PROGRAM P_Station
VAR
	_stParameter:				ST_StationParameter;
	_stHandshake:				ST_StationHandshake;
	
	_fbTakeLoad:				FB_StationTakeLoad;// 取料站
	_fbDismantling_L2:			FB_StationDismantling;// 线体2 拆解站 
	_fbDismantling_L3:			FB_StationDismantling;// 线体3 拆解站 
	_fbLine0Load:				FB_StationLine0Load;// 线体0 上料站
	_fbLine0Buffer:				FB_StationLine0Buffer;// 线体0 缓存站
	_fbLineLoad_L1:				FB_StationLineLoad;// 线体1 上料站
	_fbLineLoad_L3:				FB_StationLineLoad;// 线体3 上料站
	_fbUnloadUc_L2:				FB_StationUnloadUc;// 线体2 下UC
	_fbUnloadUc_L3:				FB_StationUnloadUc;// 线体3 下UC
	_fbUnloadElevator_L2:		FB_StationUnloadElevator;// 线体2 下工装
	_fbUnloadElevator_L3:		FB_StationUnloadElevator;// 线体3 下工装
	_fbUnloadLineUc:			FB_StationUnloadLine;//下UC 线体
	_fbUnloadLineElevator:		FB_StationUnloadLine;// 下工装线体
	_fbStationUnLoadUc_311:		FB_StationUnLoadUc_311;// 下UC 模组
		
	_vArrFbCylinder:			ARRAY[0..10] OF FB_Cylinder;// 虚拟气缸
	_vArrCylinder:				ARRAY[0..10] OF ST_Cylinder;// 虚拟气缸
	_vArrCylinderData:			ARRAY[0..10] OF ST_CylinderData;// 虚拟气缸
	_i:							INT;
	_bFistRun:					BOOL:=true;
END_VAR

GVL.stSetting.eTakeMode:=M_LoadPriority(_stParameter,GVL_Data.stRecipe);
IF _bFistRun THEN
	A_Info();
	_bFistRun:=FALSE;
END_IF


A_Handshake();// 交握

A_Virtual();// 虚拟硬件



A_TakeLoad();// 取料站

A_Dismantling_L2();// 拆解站

A_Dismantling_L3();// 拆解站

A_Line0Buffer();// 线体0 上料缓存

A_Line0Load();// 线体0 上料站

A_LineLoad_L1();// 线体1 上料

A_LineLoad_L3();// 线体3 上料

A_UnloadElevator_L2();// 线体2 下工装

A_UnloadElevator_L3();// 线体3 下工装

A_UnloadLineElevator();// 下工装 流线

A_UnLoadUc_311();// 下UC模组  紧311使用

A_UnloadLineUc();// 下UC 流线 311以为下料程序

A_UnloadUc_L2();// 线体2下UC 311以外下料程序

A_UnloadUc_L3();// 线体3 下UC 311以为下料程序

ACTION A_Dismantling_L2:
_stParameter.stLine2Dismantling.bPalletCheck1:=GVL.I.bLine2PalletCheck1;
_stParameter.stLine2Dismantling.bPalletCheck2:=GVL.I.bLine2PalletCheck2;
_stParameter.stLine2Dismantling.bPalletCheck3:=GVL.I.bLine2PalletCheck3;
_stParameter.stLine2Dismantling.fbLateral1 REF=G_arrFbCylinder[E_Cylinder.Line2OpenLateral1];
_stParameter.stLine2Dismantling.fbLateral2 REF=G_arrFbCylinder[E_Cylinder.Line2OpenLateral2];
_stParameter.stLine2Dismantling.fbLift REF= G_arrFbCylinder[E_Cylinder.Line2Lift];
_stParameter.stLine2Dismantling.fbPrevent REF= G_arrFbCylinder[E_Cylinder.Line2Prevent];
_stParameter.stLine2Dismantling.fbRotate REF= G_arrFbCylinder[E_Cylinder.Line2OpenRotate];
_stParameter.stLine2Dismantling.fbStandard1 REF= G_arrFbCylinder[E_Cylinder.Line2Standard1];
_stParameter.stLine2Dismantling.fbStandard2 REF= G_arrFbCylinder[E_Cylinder.Line2Standard2];
_stParameter.stLine2Dismantling.bClose:=GVL_Data.stRecipe.eLineClose=E_LineClose.Line2;
_stParameter.stLine2Dismantling.bCloseUnloadElevator:=FALSE;

_fbDismantling_L2(
	Enable:=TRUE,
	System:=G_stSystem , 
	Station:=G_arrStation[E_Station.Line2Dismantling] , 
	Error:=G_stError , 
	Setting:=GVL.stSetting , 
	Recipe:=GVL_Data.stRecipe , 
	Parameter:=_stParameter.stLine2Dismantling);
END_ACTION

ACTION A_Dismantling_L3:
_stParameter.stLine3Dismantling.bPalletCheck1:=GVL.I.bLine3OpenCheck1;
_stParameter.stLine3Dismantling.bPalletCheck2:=GVL.I.bLine3OpenCheck2;
_stParameter.stLine3Dismantling.bPalletCheck3:=GVL.I.bLine3OpenCheck3;
_stParameter.stLine3Dismantling.fbLateral1 REF=G_arrFbCylinder[E_Cylinder.Line3OpenLateral1];
_stParameter.stLine3Dismantling.fbLateral2 REF=G_arrFbCylinder[E_Cylinder.Line3OpenLateral2];
_stParameter.stLine3Dismantling.fbLift REF= G_arrFbCylinder[E_Cylinder.Line3OpenLift];
_stParameter.stLine3Dismantling.fbPrevent REF= G_arrFbCylinder[E_Cylinder.Line3OpenPrevent];
_stParameter.stLine3Dismantling.fbRotate REF= G_arrFbCylinder[E_Cylinder.Line3OpenRotate];
_stParameter.stLine3Dismantling.fbStandard1 REF= G_arrFbCylinder[E_Cylinder.Line3Standard1];
_stParameter.stLine3Dismantling.fbStandard2 REF= G_arrFbCylinder[E_Cylinder.Line3Standard2];
_stParameter.stLine3Dismantling.bClose:=GVL_Data.stRecipe.eLineClose=E_LineClose.Line3;
_stParameter.stLine3Dismantling.bCloseUnloadElevator:=FALSE;

_fbDismantling_L3(
	Enable:=TRUE,
	System:=G_stSystem , 
	Station:=G_arrStation[E_Station.Line3Dismantling] , 
	Error:=G_stError , 
	Setting:=GVL.stSetting , 
	Recipe:=GVL_Data.stRecipe , 
	Parameter:=_stParameter.stLine3Dismantling);
END_ACTION

ACTION A_Handshake:
_stParameter.stLine0Load.stHandshake.bRequestLine0Load:=_stParameter.stLine0Buffer.stHandshake.bRequestLine0Load;

_stParameter.stLine0Buffer.stHandshake.bRequestLine0Buffer_T:=_stParameter.stTakeLoad.stHandshake.bRequestLine0Buffer_T0;
_stParameter.stLine0Buffer.stHandshake.bResponseLine0Buffer:=_stParameter.stLine0Load.stHandshake.bResponseLine0Buffer;

_stParameter.stLine1Load.stHandshake.bRequestLineLoad_D:=_stParameter.stLine2Dismantling.stHandshake.bRequestLineLoad_D;
_stParameter.stLine1Load.stHandshake.bRequestLineLoad_P:=_stParameter.stTakeLoad.stHandshake.bRequestLineLoad_P1;
_stParameter.stLine1Load.stHandshake.bRequestLineLoad_T:=_stParameter.stTakeLoad.stHandshake.bRequestLineLoad_T1;
_stParameter.stLine1Load.stHandshake.bRequestTake_P_M:=FALSE;
_stParameter.stLine1Load.stHandshake.bResponseMachine_P:=FALSE;

_stParameter.stLine2UnloadElevator.stHandshake.bRequestElevator:=_stParameter.stLine2Dismantling.stHandshake.bRequestElevator;
_stParameter.stLine2UnloadElevator.stHandshake.bResponseElevator:=_stParameter.stUnloadLineElevator.stHandshake.bResponseUnladLine2;

_stParameter.stLine2UnloadUc.stHandshake.bResponseUnladLine:=_stParameter.stUnloadLineUc.stHandshake.bResponseUnladLine2;

_stParameter.stLine3Load.stHandshake.bRequestLineLoad_D:=_stParameter.stLine3Dismantling.stHandshake.bRequestLineLoad_D;
_stParameter.stLine3Load.stHandshake.bRequestLineLoad_P:=_stParameter.stTakeLoad.stHandshake.bRequestLineLoad_P3;
_stParameter.stLine3Load.stHandshake.bRequestLineLoad_T:=_stParameter.stTakeLoad.stHandshake.bRequestLineLoad_T3;
_stParameter.stLine3Load.stHandshake.bRequestTake_P_M:=FALSE;
_stParameter.stLine3Load.stHandshake.bResponseMachine_P:=FALSE;

_stParameter.stLine3UnloadElevator.stHandshake.bRequestElevator:=_stParameter.stLine3Dismantling.stHandshake.bRequestElevator;
_stParameter.stLine3UnloadElevator.stHandshake.bResponseElevator:=_stParameter.stUnloadLineElevator.stHandshake.bResponseUnladLine3;

_stParameter.stLine3UnloadUc.stHandshake.bResponseUnladLine:=_stParameter.stUnloadLineUc.stHandshake.bResponseUnladLine3;

_stParameter.stTakeLoad.stHandshake.bResponseTake_P1:=_stParameter.stLine1Load.stHandshake.bResponseTake_P;
_stParameter.stTakeLoad.stHandshake.bResponseTake_P3:=_stParameter.stLine3Load.stHandshake.bResponseTake_P;
_stParameter.stTakeLoad.stHandshake.bResponseTake_T0:=_stParameter.stLine0Buffer.stHandshake.bResponseTake_T;
_stParameter.stTakeLoad.stHandshake.bResponseTake_T1:=_stParameter.stLine1Load.stHandshake.bResponseTake_T;
_stParameter.stTakeLoad.stHandshake.bResponseTake_T3:=_stParameter.stLine3Load.stHandshake.bResponseTake_T;

_stParameter.stUnloadLineElevator.stHandshake.bRequestUnloadLine2:=_stParameter.stLine2UnloadElevator.stHandshake.bRequestUnline;
_stParameter.stUnloadLineElevator.stHandshake.bRequestUnloadLine3:=_stParameter.stLine3UnloadElevator.stHandshake.bRequestUnline;

_stParameter.stUnloadLineUc.stHandshake.bRequestUnloadLine2:=_stParameter.stLine2UnloadUc.stHandshake.bRequestUnloadLine;
_stParameter.stUnloadLineUc.stHandshake.bRequestUnloadLine3:=_stParameter.stLine3UnloadUc.stHandshake.bRequestUnloadLine;

_stParameter.stLine2Dismantling.stHandshake.bResponseDismantling_D:=_stParameter.stLine1Load.stHandshake.bResponseDismantling_D;
_stParameter.stLine2Dismantling.stHandshake.bResponseDismantling_E:=_stParameter.stLine2UnloadElevator.stHandshake.bResponseDismantling_E;
_stParameter.stLine3Dismantling.stHandshake.bResponseDismantling_D:=_stParameter.stLine3Load.stHandshake.bResponseDismantling_D;
_stParameter.stLine3Dismantling.stHandshake.bResponseDismantling_E:=_stParameter.stLine3UnloadElevator.stHandshake.bResponseDismantling_E;

IF GVL_Data.stRecipe.eMachineType =E_MachineType.RH311 OR GVL_Data.stRecipe.eMachineType =E_MachineType.LH311 THEN
	_stParameter.stUnloadUc_311.stHandshake.bRequestUc_L2:=_stParameter.stLine2Dismantling.stHandshake.bRequestUc;
	_stParameter.stUnloadUc_311.stHandshake.bRequestUc_L3:=_stParameter.stLine3Dismantling.stHandshake.bRequestUc;
	_stParameter.stLine2Dismantling.stHandshake.bResponseDismantling_Uc:=_stParameter.stUnloadUc_311.stHandshake.bResponseDismantling_Uc_L2;
	_stParameter.stLine3Dismantling.stHandshake.bResponseDismantling_Uc:=_stParameter.stUnloadUc_311.stHandshake.bResponseDismantling_Uc_L3;
ELSE
	_stParameter.stLine2UnloadUc.stHandshake.bRequestUc:=_stParameter.stLine2Dismantling.stHandshake.bRequestUc;
	_stParameter.stLine3UnloadUc.stHandshake.bRequestUc:=_stParameter.stLine3Dismantling.stHandshake.bRequestUc;
	_stParameter.stLine2Dismantling.stHandshake.bResponseDismantling_Uc:=_stParameter.stLine2UnloadUc.stHandshake.bResponseDismantling_Uc;
	_stParameter.stLine3Dismantling.stHandshake.bResponseDismantling_Uc:=_stParameter.stLine3UnloadUc.stHandshake.bResponseDismantling_Uc;
END_IF
END_ACTION

ACTION A_Info:
_i:=E_Station.Line0Load;
G_arrStation[_i].arrName[E_Language.Chinese]:="主流线上料工站";
G_arrStation[_i].arrName[E_Language.English]:="Line0Load";
G_arrStation[_i].arrName[E_Language.Vietnamese]:="Trạm vật liệu dòng chính";

_i:=E_Station.Line0Buffer;
G_arrStation[_i].arrName[E_Language.Chinese]:="主流线缓存工站";
G_arrStation[_i].arrName[E_Language.English]:="Line0Buffer";
G_arrStation[_i].arrName[E_Language.Vietnamese]:="Trạm bộ nhớ nhớ đường chính";

_i:=E_Station.TakeLoad;
G_arrStation[_i].arrName[E_Language.Chinese]:="上料取料工站";
G_arrStation[_i].arrName[E_Language.English]:="TakeLoad";
G_arrStation[_i].arrName[E_Language.Vietnamese]:="Nhà ga ăn uống";

_i:=E_Station.Line3Load;
G_arrStation[_i].arrName[E_Language.Chinese]:="流线3上料工站";
G_arrStation[_i].arrName[E_Language.English]:="Line3Load";
G_arrStation[_i].arrName[E_Language.Vietnamese]:="Trạm sạc 3 dòng";

_i:=E_Station.Line1Load;
G_arrStation[_i].arrName[E_Language.Chinese]:="流线2上料工站";
G_arrStation[_i].arrName[E_Language.English]:="Line1Load";
G_arrStation[_i].arrName[E_Language.Vietnamese]:="Trạm lên men dòng 2";

_i:=E_Station.Line2Dismantling;
G_arrStation[_i].arrName[E_Language.Chinese]:="流线2拆解工站";
G_arrStation[_i].arrName[E_Language.English]:="Line2Dismantling";
G_arrStation[_i].arrName[E_Language.Vietnamese]:="Trạm tháo dỡ dòng 2";

_i:=E_Station.Line3Dismantling;
G_arrStation[_i].arrName[E_Language.Chinese]:="流线3拆解工站";
G_arrStation[_i].arrName[E_Language.English]:="Line3Dismantling";
G_arrStation[_i].arrName[E_Language.Vietnamese]:="Trạm tháo dỡ dòng 3";

_i:=E_Station.Line2UnloadElevator;
G_arrStation[_i].arrName[E_Language.Chinese]:="线体2下工装";
G_arrStation[_i].arrName[E_Language.English]:="Line2UnloadElevator";
G_arrStation[_i].arrName[E_Language.Vietnamese]:="Thiết bị dây chuyền 2";

_i:=E_Station.Line3UnloadElevator;
G_arrStation[_i].arrName[E_Language.Chinese]:="线体3下工装";
G_arrStation[_i].arrName[E_Language.English]:="Line3UnloadElevator";
G_arrStation[_i].arrName[E_Language.Vietnamese]:="Dây số 3 dưới công cụ";

_i:=E_Station.Line2UnloadUc;
G_arrStation[_i].arrName[E_Language.Chinese]:="线体2 下UC";
G_arrStation[_i].arrName[E_Language.English]:="Line2UnloadUc";
G_arrStation[_i].arrName[E_Language.Vietnamese]:="Máy dò 2 ở UC";

_i:=E_Station.Line3UnloadUc;
G_arrStation[_i].arrName[E_Language.Chinese]:="线体3 下UC";
G_arrStation[_i].arrName[E_Language.English]:="Line3UnloadUc";
G_arrStation[_i].arrName[E_Language.Vietnamese]:="Máy dò 3 ở UC";

_i:=E_Station.UnloadLineUc;
G_arrStation[_i].arrName[E_Language.Chinese]:="下UC 线体";
G_arrStation[_i].arrName[E_Language.English]:="UnloadLineUc";
G_arrStation[_i].arrName[E_Language.Vietnamese]:="Ống dẫn dưới UC";

_i:=E_Station.UnloadLineElevator;
G_arrStation[_i].arrName[E_Language.Chinese]:="下工装 线体";
G_arrStation[_i].arrName[E_Language.English]:="UnloadLineElevator";
G_arrStation[_i].arrName[E_Language.Vietnamese]:="Thiết bị dây";

_i:=E_Station.UnloadUc_311;
G_arrStation[_i].arrName[E_Language.Chinese]:="下UC模组";
G_arrStation[_i].arrName[E_Language.English]:="UnloadUc_311";
G_arrStation[_i].arrName[E_Language.Vietnamese]:="Mô-đun dưới UC";
END_ACTION

ACTION A_Line0Buffer:

_stParameter.stLine0Buffer.bPlace:=GVL.I.bLine0Place;


_fbLine0Buffer(
	Enable:=TRUE,
	System:=G_stSystem , 
	Station:=G_arrStation[E_Station.Line0Buffer] , 
	Error:=G_stError , 
	Setting:=GVL.stSetting , 
	Recipe:=GVL_Data.stRecipe , 
	Parameter:=_stParameter.stLine0Buffer);
END_ACTION

ACTION A_Line0Load:
_stParameter.stLine0Load.bPartCheck:=GVL.I.bLine0Part;
_stParameter.stLine0Load.bPreventCheck:=GVL.I.bLine0Prevent;
_stParameter.stLine0Load.fbPart REF= G_arrFbCylinder[E_Cylinder.Line0Part];
_stParameter.stLine0Load.fbPrevent REF= G_arrFbCylinder[E_Cylinder.Line0Prevent];

_fbLine0Load(
	Enable:=TRUE,
	System:=G_stSystem , 
	Station:=G_arrStation[E_Station.Line0Load] , 
	Error:=G_stError , 
	Setting:=GVL.stSetting , 
	Recipe:=GVL_Data.stRecipe , 
	Parameter:=_stParameter.stLine0Load);
END_ACTION

ACTION A_LineLoad_L1:
_stParameter.stLine1Load.bIsClosed:=GVL_Data.stRecipe.eLoadClose=E_LoadClose.Line1;
_stParameter.stLine1Load.bIsPlacing:=GVL.stSetting.eTakeModeBuffer=E_TakeMode.Place1;
_stParameter.stLine1Load.bIsTaking:=GVL.stSetting.eTakeModeBuffer=E_TakeMode.Take1;
_stParameter.stLine1Load.bPalletCheck1:=GVL.I.bLine1PalletCheck1;
_stParameter.stLine1Load.bPalletCheck2:=GVL.I.bLine1PalletCheck2;
_stParameter.stLine1Load.bPalletCheck3:=GVL.I.bLine1PalletCheck3;
_stParameter.stLine1Load.fbAdjust1 REF= G_arrFbCylinder[E_Cylinder.Line1Adjust1];
_stParameter.stLine1Load.fbElevator REF= G_arrFbCylinder[E_Cylinder.Line1Elevator];
_stParameter.stLine1Load.fbLift REF= G_arrFbCylinder[E_Cylinder.Line1Lift];
_stParameter.stLine1Load.fbPrevent REF= G_arrFbCylinder[E_Cylinder.Line1Prevent];
_stParameter.stLine1Load.fbRotate REF= G_arrFbCylinder[E_Cylinder.Line1Rotate];
_stParameter.stLine1Load.bManualLoad:=FALSE;
_fbLineLoad_L1(
	Enable:=true,
	System:=G_stSystem , 
	Station:=G_arrStation[E_Station.Line1Load] , 
	Error:=G_stError , 
	Setting:=GVL.stSetting , 
	Recipe:=GVL_Data.stRecipe , 
	Parameter:=_stParameter.stLine1Load);
END_ACTION

ACTION A_LineLoad_L3:
_stParameter.stLine3Load.bIsClosed:=FALSE;
_stParameter.stLine3Load.bIsPlacing:=GVL.stSetting.eTakeModeBuffer=E_TakeMode.Place3Load;
_stParameter.stLine3Load.bIsTaking:=GVL.stSetting.eTakeModeBuffer=E_TakeMode.Take3Load;
_stParameter.stLine3Load.bPalletCheck1:=GVL.I.bLine3PalletCheck1;
_stParameter.stLine3Load.bPalletCheck2:=GVL.I.bLine3PalletCheck2;
_stParameter.stLine3Load.bPalletCheck3:=GVL.I.bLine3PalletCheck3;
_stParameter.stLine3Load.fbAdjust1 REF= _vArrFbCylinder[0];
_stParameter.stLine3Load.fbElevator REF=_vArrFbCylinder[1];
_stParameter.stLine3Load.fbLift REF= G_arrFbCylinder[E_Cylinder.Line3LoadLift];
_stParameter.stLine3Load.fbPrevent REF= G_arrFbCylinder[E_Cylinder.Line3LoadPrevent];
_stParameter.stLine3Load.fbRotate REF= G_arrFbCylinder[E_Cylinder.Line3LoadRotate];
_stParameter.stLine3Load.bManualLoad:=FALSE;

_fbLineLoad_L3(
	Enable:=TRUE,
	System:=G_stSystem , 
	Station:=G_arrStation[E_Station.Line3Load] , 
	Error:=G_stError , 
	Setting:=GVL.stSetting , 
	Recipe:=GVL_Data.stRecipe , 
	Parameter:=_stParameter.stLine3Load);
END_ACTION

ACTION A_TakeLoad:
_stParameter.stTakeLoad.fbTakeClamp REF= G_arrFbCylinder[E_Cylinder.TakeClamp];
_stParameter.stTakeLoad.fbTakeLift1 REF= G_arrFbCylinder[E_Cylinder.TakeLift1];
_stParameter.stTakeLoad.fbTakeLift2 REF= G_arrFbCylinder[E_Cylinder.TakeLift2];
_stParameter.stTakeLoad.fbTakeY REF= G_arrFbAxis[E_Axis.TakeY];
_stParameter.stTakeLoad.fbTakeZ REF= G_arrFbAxis[E_Axis.TakeZ];

_fbTakeLoad(
	Enable:=TRUE,
	System:=G_stSystem , 
	Station:=G_arrStation[E_Station.TakeLoad] , 
	Error:=G_stError , 
	Setting:=GVL.stSetting , 
	Recipe:=GVL_Data.stRecipe , 
	Parameter:=_stParameter.stTakeLoad);
END_ACTION

ACTION A_UnloadElevator_L2:
_stParameter.stLine2UnloadElevator.bFrockElevator1NoneCheck:=GVL.I.bFrockElevator1NoneCheck;
_stParameter.stLine2UnloadElevator.fbFrockElevator REF= G_arrFbCylinder[E_Cylinder.FrockElevator1];
_stParameter.stLine2UnloadElevator.fbFrockPush REF= G_arrFbCylinder[E_Cylinder.FrockPush1];
_stParameter.stLine2UnloadElevator.fbFrockRotateDown REF= G_arrFbCylinder[E_Cylinder.FrockRotateDown1];
_stParameter.stLine2UnloadElevator.bManualUnload:=FALSE;


_fbUnloadElevator_L2(
	Enable:=TRUE,
	System:=G_stSystem , 
	Station:=G_arrStation[E_Station.Line2UnloadElevator] , 
	Error:=G_stError , 
	Setting:=GVL.stSetting , 
	Recipe:=GVL_Data.stRecipe , 
	Parameter:=_stParameter.stLine2UnloadElevator);
END_ACTION

ACTION A_UnloadElevator_L3:

_stParameter.stLine3UnloadElevator.bFrockElevator1NoneCheck:=GVL.I.bFrockElevator2NoneCheck;
_stParameter.stLine3UnloadElevator.fbFrockElevator REF= G_arrFbCylinder[E_Cylinder.FrockElevator2];
_stParameter.stLine3UnloadElevator.fbFrockPush REF= G_arrFbCylinder[E_Cylinder.FrockPush2];
_stParameter.stLine3UnloadElevator.fbFrockRotateDown REF= G_arrFbCylinder[E_Cylinder.FrockRotateDown2];
_stParameter.stLine3UnloadElevator.bManualUnload:=FALSE;

_fbUnloadElevator_L3(
	Enable:=TRUE,
	System:=G_stSystem , 
	Station:=G_arrStation[E_Station.Line3UnloadElevator] , 
	Error:=G_stError , 
	Setting:=GVL.stSetting , 
	Recipe:=GVL_Data.stRecipe , 
	Parameter:=_stParameter.stLine3UnloadElevator);
END_ACTION

ACTION A_UnloadLineElevator:
_stParameter.stUnloadLineElevator.bBeltDone:=GVL.I.bFrockBeltDone;
_stParameter.stUnloadLineElevator.bBeltNoneCheck:=GVL.I.bFrockBeltNoneCheck3;
_stParameter.stUnloadLineElevator.bCheck1:=GVL.I.bFrockBeltNoneCheck1;
_stParameter.stUnloadLineElevator.bCheck2:=GVL.I.bFrockBeltNoneCheck2;
_stParameter.stUnloadLineElevator.fbDrive REF= G_arrFbCylinder[E_Cylinder.FrockBelt];
_stParameter.stUnloadLineElevator.fbLineAxis REF= GVL.arrFbLine[E_Line.UnloadElevator];
_stParameter.stUnloadLineElevator.bManualUnload:=FALSE;

_fbUnloadLineElevator(
	Enable:=TRUE,
	System:=G_stSystem , 
	Station:=G_arrStation[E_Station.UnloadLineElevator] , 
	Error:=G_stError , 
	Setting:=GVL.stSetting , 
	Recipe:=GVL_Data.stRecipe , 
	Parameter:=_stParameter.stUnloadLineElevator);
END_ACTION

ACTION A_UnloadLineUc:
_stParameter.stUnloadLineUc.bBeltDone:=GVL.I.bUcBeltDone;
_stParameter.stUnloadLineUc.bBeltNoneCheck:=GVL.I.bUcBeltNoneCheck;
_stParameter.stUnloadLineUc.bCheck1:=GVL.I.bUcCheck2;
_stParameter.stUnloadLineUc.bCheck2:=GVL.I.bUcCheck3;
_stParameter.stUnloadLineUc.fbDrive REF= G_arrFbCylinder[E_Cylinder.UcDrive];
_stParameter.stUnloadLineUc.fbLineAxis REF= GVL.arrFbLine[E_Line.UnloadUC];
_stParameter.stUnloadLineUc.bManualUnload:=FALSE;

_fbUnloadLineUc(
	Enable:=NOT(GVL_Data.stRecipe.eMachineType=E_MachineType.LH311 OR GVL_Data.stRecipe.eMachineType=E_MachineType.RH311),
	System:=G_stSystem , 
	Station:=G_arrStation[E_Station.UnloadLineUc] , 
	Error:=G_stError , 
	Setting:=GVL.stSetting , 
	Recipe:=GVL_Data.stRecipe , 
	Parameter:=_stParameter.stUnloadLineUc);
END_ACTION

ACTION A_UnLoadUc_311:
_stParameter.stUnloadUc_311.bUcCheck1:=GVL.I.bUcCheck1;
_stParameter.stUnloadUc_311.fbAxisY REF= G_arrFbAxis[E_Axis.UC_Y];
_stParameter.stUnloadUc_311.fbClamp REF= G_arrFbCylinder[E_Cylinder.UcClamp];
_stParameter.stUnloadUc_311.fbLift REF= G_arrFbCylinder[E_Cylinder.UcLift];
_stParameter.stUnloadUc_311.fbSwing REF= G_arrFbCylinder[E_Cylinder.UcSwing];

_fbStationUnLoadUc_311(
	Enable:=GVL_Data.stRecipe.eMachineType=E_MachineType.LH311 OR GVL_Data.stRecipe.eMachineType=E_MachineType.RH311,
	System:=G_stSystem , 
	Station:=G_arrStation[E_Station.UnloadUc_311] , 
	Error:=G_stError , 
	Setting:=GVL.stSetting , 
	Recipe:=GVL_Data.stRecipe , 
	Parameter:=_stParameter.stUnloadUc_311);
END_ACTION

ACTION A_UnloadUc_L2:
_stParameter.stLine2UnloadUc.fbClamp REF= G_arrFbCylinder[E_Cylinder.UcClamp1];
_stParameter.stLine2UnloadUc.fbLift REF= G_arrFbCylinder[E_Cylinder.UcLift1];
_stParameter.stLine2UnloadUc.fbRotate REF= G_arrFbCylinder[E_Cylinder.UcRotate1];

_fbUnloadUc_L2(
	Enable:=NOT(GVL_Data.stRecipe.eMachineType=E_MachineType.LH311 OR GVL_Data.stRecipe.eMachineType=E_MachineType.RH311),
	System:=G_stSystem , 
	Station:=G_arrStation[E_Station.Line2UnloadUc] , 
	Error:=G_stError , 
	Setting:=GVL.stSetting , 
	Recipe:=GVL_Data.stRecipe , 
	Parameter:=_stParameter.stLine2UnloadUc);
END_ACTION

ACTION A_UnloadUc_L3:
_stParameter.stLine3UnloadUc.fbClamp REF= G_arrFbCylinder[E_Cylinder.UcClamp2];
_stParameter.stLine3UnloadUc.fbLift REF= G_arrFbCylinder[E_Cylinder.UcLift2];
_stParameter.stLine3UnloadUc.fbRotate REF= G_arrFbCylinder[E_Cylinder.UcRotate2];

	
_fbUnloadUc_L3(
	Enable:=NOT(GVL_Data.stRecipe.eMachineType=E_MachineType.LH311 OR GVL_Data.stRecipe.eMachineType=E_MachineType.RH311),
	System:=G_stSystem , 
	Station:=G_arrStation[E_Station.Line3UnloadUc] , 
	Error:=G_stError , 
	Setting:=GVL.stSetting , 
	Recipe:=GVL_Data.stRecipe , 
	Parameter:=_stParameter.stLine3UnloadUc);
END_ACTION

ACTION A_Virtual:
FOR _i:=0 TO 10 BY 1 DO
	_vArrCylinder[_i].stInput.bHome:=_vArrCylinder[_i].stOutput.bHome;
	_vArrCylinder[_i].stInput.bWork:=_vArrCylinder[_i].stOutput.bWork;
	_vArrFbCylinder[_i](System:=G_stSystem , Cylinder:=_vArrCylinder[_i] , Data:=_vArrCylinderData[_i] , Error:=G_stError );
END_FOR
END_ACTION

METHOD M_LoadPriority : E_TakeMode
VAR_INPUT
	Parameter:		 REFERENCE TO ST_StationParameter;
	Recipe:			 REFERENCE TO ST_Recipe;	
END_VAR
VAR
	_iTemp:					INT;
END_VAR
M_LoadPriority:=E_TakeMode.None;


IF Parameter.stTakeLoad.eState=E_StationState.Done THEN
	IF Parameter.stLine1Load.eState=E_StationState.Load AND Recipe.eLineClose<>E_LineClose.Line2 THEN
		M_LoadPriority:=E_TakeMode.Place1;
	END_IF
	IF Parameter.stLine3Load.eState=E_StationState.Load AND Recipe.eLineClose<>E_LineClose.Line3 THEN
		M_LoadPriority:=E_TakeMode.Place3Load;
	END_IF
END_IF

IF Parameter.stTakeLoad.eState=E_StationState.Load THEN
	IF Parameter.stLine3Load.eState=E_StationState.Done AND Recipe.eLineClose=E_LineClose.Line3 THEN
		M_LoadPriority:=E_TakeMode.Take3Load;
	END_IF
	CASE Recipe.eLoadPriority OF
	E_LoadPriority.None,E_LoadPriority.Line0:
		IF Parameter.stLine1Load.eState=E_StationState.Done AND ((Parameter.stLine3Dismantling.eState=E_StationState.Load AND Parameter.stLine3Load.eState=E_StationState.Load) OR Recipe.eLineClose=E_LineClose.Line2) THEN
			M_LoadPriority:=E_TakeMode.Take1;
		END_IF
		IF Parameter.stLine0Buffer.eState=E_StationState.Done THEN
			M_LoadPriority:=E_TakeMode.Take0;
		END_IF
	E_LoadPriority.Line1:
		IF Parameter.stLine0Buffer.eState=E_StationState.Done THEN
			M_LoadPriority:=E_TakeMode.Take0;
		END_IF
		IF Parameter.stLine1Load.eState=E_StationState.Done AND (Parameter.stLine3Load.eState=E_StationState.Load OR Recipe.eLineClose=E_LineClose.Line2) THEN
			M_LoadPriority:=E_TakeMode.Take1;
		END_IF
	END_CASE
END_IF
END_METHOD

END_PROGRAM

(* stored: Version 1.1.0.1, ProductVersion 3.1.4024.3
   POU P_Station: Id {79a78cd0-f841-421e-a4ef-6ebd8d61ff55}, SpecialFunc None
   Action A_Dismantling_L2: Id {b01f12b6-60a3-4639-b368-e374f1faa4f5}
   Action A_Dismantling_L3: Id {06e81362-3cd9-4009-9cc8-dae5d0f41afb}
   Action A_Handshake: Id {4cd92d19-1b07-440d-87b6-562e0563fd0c}
   Action A_Info: Id {e3cbee2e-0c6d-4e1e-9333-7eeb974869ab}
   Action A_Line0Buffer: Id {3c682dc6-e395-440e-8dfc-056387168c36}
   Action A_Line0Load: Id {dba4453f-7678-4827-939f-b06b9b20f201}
   Action A_LineLoad_L1: Id {d92e3f6f-3284-41b5-b4d6-24b94807dc78}
   Action A_LineLoad_L3: Id {b507f1d5-e932-43d6-abaa-167c55cb752d}
   Action A_TakeLoad: Id {aabca987-a068-415b-aaa7-c4e58e7fb99d}
   Action A_UnloadElevator_L2: Id {429ef40b-80da-4ad2-89d3-54f75010941e}
   Action A_UnloadElevator_L3: Id {e148bbd6-1eb7-4ca1-af65-fb7edc507d40}
   Action A_UnloadLineElevator: Id {435894e7-c2dc-4c13-b90c-d062ebb83a2a}
   Action A_UnloadLineUc: Id {83d00882-42dd-4202-9c11-b79a6589fac3}
   Action A_UnLoadUc_311: Id {60121d26-0a8f-4cdd-ab14-c744b69a556d}
   Action A_UnloadUc_L2: Id {a65e0f00-d046-4752-bae9-0e435ea1babb}
   Action A_UnloadUc_L3: Id {af63726c-2292-41d9-b43d-84bf4ea87ffa}
   Action A_Virtual: Id {9ea1df27-9ec0-40a8-871b-324c9f2f1f9b}
   Method M_LoadPriority: Id {ab313c0c-22fc-4a11-84d5-bc2b1c22c5cb} *)
